FUNCTION_BLOCK Q_LineAttributes (* Command change line attributes ( Part 6 - F.30 ) *)
  (* Standard: ISO 11783-6; Description: Copyright (c) 2022 HR Agrartechnik GmbH This program and the accompanying materials are made available under the terms of the Eclipse Public License 2.0 which is available at https://www.eclipse.org/legal/epl-2.0/ SPDX-License-Identifier: EPL-2.0 see Description Tab *)
  (* Version 1.0, 2022-07-08, Franz Höpfinger, HR Agrartechnik GmbH *)
  (* Documentation:
  Command change line attributes ( Part 6 - F.30 )
   This command is used to change the line attributes in a line attributes object.
   param[in] {objectID, uint16_t}
   Object ID
   param[in] {colour, uint8_t}
   New line colour (see Part 6 - A.3)
   param[in] {width, uint8_t}
   New line width (see Part 6 - B.14.3)
   param[in] {lineArtBitmask, uint16_t}
   New line art (see Part 6 - B.14.3)
   Return Values: 
   int16_t
    - VT_E_NO_ERR (0) - OK
   - VT_E_OVERFLOW (-6) - buffer overflow
   - VT_E_NOACT (-8) - Command not possible in current state
   - VT_E_NO_INSTANCE (-21) - No VT client available
   - VT_E_ISO_INSTANCE_INVALID (-129) - Identifier for instance (connection) invalid
   - VT_E_NOT_ALIVE (-130) - Identifier for instance valid, but VT Dead.
  *)
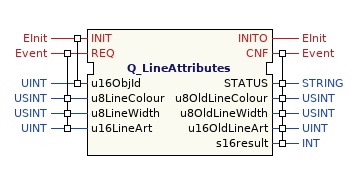
  EVENT_INPUT
    INIT : EInit WITH u16ObjId; (* Service Initialization *)
    REQ WITH u8LineColour, u8LineWidth, u16LineArt; (* Service Request *)
  END_EVENT
  EVENT_OUTPUT
    INITO : EInit; (* Initialization Confirm *)
    CNF WITH STATUS, s16result, u8OldLineColour, u8OldLineWidth, u16OldLineArt; (* Confirmation of Requested Service *)
  END_EVENT
  VAR_INPUT
    u16ObjId : UINT; (* Object ID *)
    u8LineColour : USINT; (* New line colour *)
    u8LineWidth : USINT; (* New line width (see Part 6 - B.14.3) *)
    u16LineArt : UINT; (* New line art (see Part 6 - B.14.3) *)
  END_VAR
  VAR_OUTPUT
    STATUS : STRING; (* Service Status *)
    u8OldLineColour : USINT; (* Old line colour *)
    u8OldLineWidth : USINT; (* Old line width (see Part 6 - B.14.3) *)
    u16OldLineArt : UINT; (* Old line art (see Part 6 - B.14.3) *)
    s16result : INT; (* retval see description *)
  END_VAR
END_FUNCTION_BLOCK
